// TIA Portal project "260610_V006_S7300_3BänderAblaufsteuerungBeton" (V17)

(* hardware
DEVICE "S7-300/ET200M-Station_1"  S7-300 station
   slot 0: "Profilschiene_0"  Rail  6ES7 390-1***0-0AA0
   slot 2: "PLC_1"  CPU 314C-2 DP  6ES7 314-6CH04-0AB0  V3.3
      slot 0: "MPI-Schnittstelle_1"  MPI
      slot 1: "DP-Schnittstelle_1"  DP
      slot 2: "DI 24/DO 16_1"  DI24/DO16
      slot 3: "AI 5/AO 2_1"  AI5/AO2
      slot 4: "Zählen_1"  Counter
      slot 5: "Positionieren_1"  Positioning
   slot 4: "DI 16/DO 16x24VDC/0.5A_1"  DI16/DO16 x 24V / 0.5A  6ES7 323-1BL00-0AA0
   slot 5: "DI 16x24VDC_1"  DI16 x 24VDC  6ES7 321-1BH02-0AA0
   slot 6: "CP 342-5_1"  CP 342-5  6GK7 342-5DA03-0XE0  V6.0
   slot 7: "CP 343-1_1"  CP 343-1  6GK7 343-1EX30-0XE0  V3.0
*)

// ===== PLC "PLC_1"  CPU 314C-2 DP =====

VAR_GLOBAL   // PLC tag table "Standard-Variablentabelle"
   "EB124_125" AT %EW124 : Word;
   "AB124_125" AT %AW124 : Word;
   "RV_scale" AT %MW118 : Word;
   "kanal0 NormwertAE" AT %MD120 : Real;
   "Kanal0" AT %EW752 : Int;
END_VAR

ORGANIZATION_BLOCK "Main"   // OB1, FBD
TITLE = "Main Program Sweep (Cycle)"
{ S7_Optimized_Access := 'FALSE' }
VERSION : 0.1
   VAR_TEMP
      OB1_EV_CLASS : Byte;   // Bits 0-3 = 1 (Coming event), Bits 4-7 = 1 (Event class 1)
      OB1_SCAN_1 : Byte;   // 1 (Cold restart scan 1 of OB 1), 3 (Scan 2-n of OB 1)
      OB1_PRIORITY : Byte;   // Priority of OB Execution
      OB1_OB_NUMBR : Byte;   // 1 (Organization block 1, OB1)
      OB1_RESERVED_1 : Byte;   // Reserved for system
      OB1_RESERVED_2 : Byte;   // Reserved for system
      OB1_PREV_CYCLE : Int;   // Cycle time of previous OB1 scan (milliseconds)
      OB1_MIN_CYCLE : Int;   // Minimum cycle time of OB1 (milliseconds)
      OB1_MAX_CYCLE : Int;   // Maximum cycle time of OB1 (milliseconds)
      OB1_DATE_TIME : Date_And_Time;   // Date and time OB1 started
      tempFalse : Bool;
   END_VAR
BEGIN

REGION Network 1
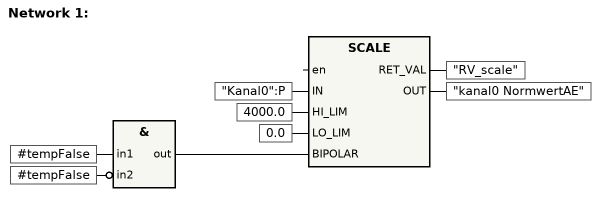
   "RV_scale" := SCALE(IN := "Kanal0":P,
                       HI_LIM := 4000.0,
                       LO_LIM := 0.0,
                       BIPOLAR := #tempFalse AND NOT #tempFalse,
                       OUT => "kanal0 NormwertAE");
END_REGION

REGION Network 2 (STL)
         L     "EB124_125";

         BEU;
END_REGION
END_ORGANIZATION_BLOCK